TYPE "UDT_ZC_DISP_AGRUP"
VERSION : 0.1
   STRUCT
      AlgunaEnManual : Bool := TRUE;   // Algun dispositivo en manual
      AlgunaAlarma : Bool := FALSE;   // Algun dispositivo en alarma
      NuevaAlarma : Bool := FALSE;   // Nueva alarma
   END_STRUCT;

END_TYPE

